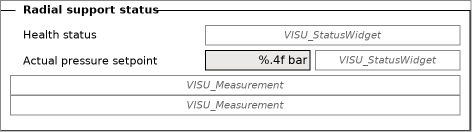
VISUALIZATION VISU_M1RadialSupportStatus  // 472x132
VAR_IN_OUT
	ref : M1RadialSupport;
    widget : M1RadialSupportWidget;
END_VAR
    Rectangle (205,50 105x20), "%.4f bar", text variable: ref.actualPressureSetpoint.bar.value
    Label (20,51 145x20), "Actual pressure setpoint"
    Frame (205,25 255x20)
        shows VISU_StatusWidget(widget := widget.actualStatus)
    Label (20,25 185x20), "Health status"
    Frame (10,75 450x20)
        shows VISU_Measurement(widget := widget.regulatorPressure)
    Frame (10,95 450x20)
        shows VISU_Measurement(widget := widget.mirrorPressure)
    Frame (315,50 145x20)
        shows VISU_StatusWidget(widget := widget.operatingStatus)
    Label (20,0 200x20), "Radial support status"
    Line (0,10) (15,10)
        p2175578022: widget.actualStatus.color.bg
    Line (155,10) (470,10)
        p2175578022: widget.actualStatus.color.bg
    Line (0,130) (470,130)
        p2175578022: widget.actualStatus.color.bg
    Line (470,130) (470,10)
        p2175578022: widget.actualStatus.color.bg
    Line (0,130) (0,10)
        p2175578022: widget.actualStatus.color.bg
END_VISUALIZATION

(* stored: Version 1.1.0.1, ProductVersion 3.1.4019.2
   Visu VISU_M1RadialSupportStatus: Id {ad233d1c-3f91-4593-be82-19cec3975bfd} *)
